PROGRAM Visu
VAR
	bStartTL1 : BOOL;
	bStartTL2 : BOOL;
	bStartTL3 : BOOL;
END_VAR

END_PROGRAM

(* stored: Version 1.1.0.1, ProductVersion 3.1.4024.2
   POU Visu: Id {653c8121-0635-4deb-8265-58d9590949a7}, SpecialFunc None *)
